(* IEC 61131-3 sources: xpxp/deepseek-coder-6.7b, 22 files *)

(* ---- 18.st ---- *)
plc
FUNCTION FC1003
	VAR_INPUT
		IN_R : REAL; (* Input real number *)
		IN_MAX, IN_MIN : REAL; (* Input min/max range for conversion *)
		OUT_MAX, OUT_MIN : REAL; (* Output min/max range for conversion *)
	END_VAR

	VAR_OUTPUT
		OUT_R : REAL; (* Result real number *)
		FEH : BOOL; (* Error flag indicating out-of-range *)
	END<｜begin▁of▁sentence｜>END_VAR

	VAR_TEMP
		DIFF1, DIFF2 : REAL; (* Temporary variables for scale calculation *)
		scl_factor : REAL; (* Scaling factor *)
		rescaled : REAL; (* Input rescaled to original range *)
	END<｜begin▁of▁sentence｜>END_VAR

	// Calculate scaling factor
	scl_factor := (OUT_MAX - OUT_MIN) / (IN_MAX - IN_MIN);

	// Rescale input value from its original range into the new one
	rescaled := scl_factor * (IN_R - IN_MIN) + OUT_MIN;

	(* Check if result is within output range *)
	IF ((rescaled < OUT_MIN) OR (rescaled > OUT_MAX)) THEN
		// If not, set error flag and return
		FEH := TRUE;
	ELSE
		OUT_R := rescaled;
	END_IF;

	// Return result and error flag to caller
	RETURN;
END_FUNCTION

(* ---- 22.st ---- *)
PLC_Programming
FUNCTION BLOCK fbMoveArm
VAR_INPUT
	MoveToWorkCmd : BOOL; // Move towards Work position command
	MoveToHomeCmd : BOOL; // Move towards Home position command
	AtWorkSensor : BOOL;  // Sensor indicating the arm is at the Work position
	AtHomeSensor : BOOL;  // Sensor indicating the arm is at the Home position
	MovementPermitted : BOOL; // Global safety signal allowing movement
END_VAR

VAR_OUTPUT
	MotorForward : BOOL; // Controls motor to move towards Work position
	MotorReverse : BOOL; // Controls motor to move towards Home position
END_VAR

// Store the previous command status for cancellation logic
VAR
	PrevMoveToWorkCmd : BOOL;
	PrevMoveToHomeCmd : BOOL;
END_VAR

IF MovementPermitted THEN
	// Cancel movement in opposite direction if current command is pressed
	MotorForward := (NOT PrevMoveToHomeCmd) AND MoveToWorkCmd;
	MotorReverse := (NOT PrevMoveToWorkCmd) AND MoveToHomeCmd;

	// Remember the status of current commands for cancellation logic
	PrevMoveToWorkCmd := MoveToWorkCmd;
	PrevMoveToHomeCmd := MoveToHomeCmd;
ELSE // If movement is not permitted, stop motors immediately
	MotorForward := FALSE;
	MotorReverse := FALSE;
END_IF

// Stop motor if at the target position
MotorForward := MotorForward AND (NOT AtWorkSensor);
MotorReverse := MotorReverse AND (NOT AtHomeSensor);
END_FUNCTION_BLOCK

(* ---- 1.st ---- *)
plc
PROGRAM MyProgram
VAR
    // Global Variables
	xAllOn : BOOL;
	xAlarm1: BOOL := FALSE;
	xAlarm2: BOOL := FALSE;
	xAllOff: BOOL;
END_VAR

// Initialize your variables here (if any)
// For example, xAllOn := TRUE;

FUNCTION_BLOCK FbUpdateAlarms
VAR_INPUT
    inAlarm1: BOOL;
    inAlarm2: BOOL;
END_VAR
VAR_OUTPUT
    outAlarm1 : BOOL;
    outAlarm2 : BOOL;
END_VAR
BEGIN
    // Update the alarms based on the input values
    IF (inAlarm1 = TRUE) THEN
        outAlarm1 := TRUE;
    END_IF;

    IF (inAlarm2 = TRUE) THEN
        outAlarm2 := TRUE;
    END_IF;
END_FUNCTION_BLOCK

// Create a new FB for updating alarms
FbUpdateAlarms(xAllOn, xAllOff, xAlarm1, xAlarm2);

(* ---- 11.st ---- *)
plc
PROGRAM SignFunction
VAR
    x : REAL; // input variable
END_VAR

FUNCTION_BLOCK FB_Sign
VAR_INPUT
    a : REAL;
END_VAR

VAR_OUTPUT
    result : INT;
END_VAR
END_FUNCTION_BLOCK

// Main function block where the program starts
FUNCTION_BLOCK FB_Main
VAR_INPUT
    x : REAL; // input variable
END_VAR

VAR_OUTPUT
    signValue : INT;
END_VAR
END_FUNCTION_BLOCK

(* ---- 19.st ---- *)
plaintext
PROGRAM Program1

FUNCTION_BLOCK FB1005
    (* VARIABLES DECLARATION *)
    VAR_INPUT
        START : BOOL;   // Start input for measurement cycle
        DICKE, V_MAX, V_MIN: REAL;  // Plate thickness and tolerance band values
    END_VAR

    VAR_OUTPUT
        D_MAX, D_MIN: REAL;  // Outputs for the maximum (D_MAX) and minimum (D_MIN) plate thickness
        P1: BOOL;   // Reject light P1 output
    END_VAR

    VAR
        FO: BOOL;  // Flag to indicate if a measurement is currently ongoing
        M_MAX, M_MIN : REAL;  // Maximum and minimum plate thickness during measurement cycle
    END_VAR
END_FUNCTION_BLOCK

(* FUNCTION BLOCK IMPLEMENTATION *)
PROGRAM Main
BEGIN
    (* Initialization of function block FB1005 *)
    FB1005(START := FALSE, DICKE := 0.0, V_MAX := 0.0, V_MIN := 0.0);

    (* Program main loop *)
    WHILE TRUE DO
        IF FB1005.START = TRUE THEN
            FO := TRUE;   // Start a measurement cycle

            M_MAX := DICKE;  // Initialize maximum plate thickness to current measured value
            M_MIN := DICKE;  // Initialize minimum plate thickness to current measured value
        END_IF;

        IF FO = TRUE THEN    // If a measurement cycle is ongoing
            FB1005.D_MAX := M_MAX;   // Output the maximum plate thickness
            FB1005.D_MIN := M_MIN;   // Output the minimum plate thickness

            IF (M_MAX > V_MAX) OR (M_MIN < V_MIN) THEN  // If current measurement violates tolerance band
                FB1005.P1 := TRUE;    // Switch on reject light P1
            END_IF;
        ELSE   // Else if no measurement cycle is ongoing, reset outputs
            FB1005.D_MAX := 0.0;
            FB1005.D_MIN := 0.0;
            FB1005.P1 := FALSE;
        END_IF;

        // Update maximum and minimum plate thickness for next measurement cycle
        M_MAX := MAX(M_MAX, DICKE);
        M_MIN := MIN(M_MIN, DICKE);
    END_WHILE;
END PROGRAM

(* ---- 20.st ---- *)
plaintext
PROGRAM MyProgram
VAR
    // Instantiate our interlock function block
    InterlockFb : INTERLOCK;

    // Declare the inputs I1, I2 and TL
    I1 : BOOL;
    I2 : BOOL;
    TL : TIME := T#5s;  // Dead time of 5 seconds
END_VAR

FUNCTION_BLOCK INTERLOCK
    VAR_INPUT
        I1 : BOOL;
        I2 : BOOL;
        TL : TIME;
    END_VAR

    VAR_OUTPUT
        Q1 : BOOL;
        Q2 : BOOL;
    END_VAR

    VAR
        T1 : TOF; // Time of FAlse for Q1
        T2 : TOF; // Time of False for Q2
    END_VAR

    IF I1 AND NOT Q1 THEN // If input is TRUE and output is FALSE, set Q1 to TRUE after dead time TL
        Q1(PT:=TL);
    ELSE
        Q1 := FALSE; // Reset Q1 if inputs are FALSE or already at TRUE for longer than deadtime TL
    END_IF;

    IF I2 AND NOT Q2 THEN // Same logic applies to Q2
        Q2(PT:=TL);
    ELSE
        Q2 := FALSE;
    END_IF;
END_FUNCTION_BLOCK

// Connections between PLC inputs and FB variables
I1 := DI[0]; // Connecting a digital input DI[0] to I1
I2 := DI[1]; // Connecting another digital input DI[1] to I2

InterlockFb(I1:=I1, I2:=I2, TL:=TL);  // Instantiating the FB in a way that its inputs correspond to our declared variables

Q1 := InterlockFb.Q1;  // Connecting the output Q1 of the function block back to an output on the PLC
Q2 := InterlockFb.Q2;  // Same logic applies for Q2
END_PROGRAM

(* ---- 21.st ---- *)
plc
FUNCTION_BLOCK BURNER
VAR_INPUT
    IN  : BOOL;
    STAGE2  : BOOL;
    OVER_TEMP  : BOOL;
    OIL_TEMP : BOOL := TRUE;
    FLAME  : BOOL;
    RST  : BOOL;
    RST_TIMER  : BOOL;
    PRE_HEAT_TIME  : TIME := t#5s;
    PRE_VENT_TIME : TIME := t#15s;
    PRE_IGNITE_TIME  : TIME := t#15s;
    POST_IGNITE_TIME  : TIME := t#25s;
    STAGE2_DELAY : TIME := t#10s;
    SAFETY_TIME  : TIME := t#5s;
    LOCKOUT_TIME : TIME := t#10s;
    MULTIPLE_IGNITION  : BOOL := TRUE;
    KW1  : REAL;
    KW2  : REAL;
END_VAR
VAR_OUTPUT
    MOTOR  : BOOL;
    COIL1  : BOOL;
    COIL2  : BOOL;
    PRE_HEAT  : BOOL;
    IGNITE  : BOOL;
    FAIL  : BOOL;
    KWH : REAL;
    STATUS  : BYTE;
END_VAR
VAR_IN_OUT
    RUNTIME1  : UDINT;
    RUNTIME2  : UDINT;
    CYCLES  : UDINT;
END_VAR
VAR
    state  : INT := 0; (* State variable to hold the current state of BURNER *)
    last  : TIME; (* Last cycle time *)
    tx  : TIME; (* Timeout *)
    last_change  : TIME; (* Last change in input *)
    timer1  : TON; (* Timer for PRE_HEAT_TIME *)
    timer2  : TON; (* Timer for other times *)
    oil_temp_last  : BOOL; (* Last state of OIL_TEMP *)
    cycles2  : UDINT; (* Number of cycles since RST was TRUE *)
END_VAR
END_FUNCTION_BLOCK

(* ---- 10.st ---- *)
plc
PROGRAM Sigmoid
VAR
    // Input variable for input data X
    input : REAL; END_VAR

    // Output variable for result Y
    output : REAL; END_VAR
END_VAR
    // Variables used in the sigmoid calculation
    temp1, temp2: REAL;
    numerator: LREAL;
    denominator: LREAL;

BEGIN
    // Calculation of sigmoid value
    temp1 := EXP(input);
    temp2 := 1 + temp1;

    numerator := temp1;
    denominator := temp2 * temp2;

    output := numerator / denominator;
END_PROGRAM

(* ---- 12.st ---- *)
plc
PROGRAM HyperbolicSine
    VAR
        X : REAL; (* Input variable *)
        Temp1, Temp2 : REAL; (* Temporary variables to hold intermediate results *)
        Result : REAL; (* Output variable for the result *)
    END_VAR

    (* Hyperbolic Sine Function using Exponential Function *)
    HSINE := EXP(X) / (EXP(X) + EXP(-X)) * 2.0;
END_PROGRAM

(* ---- 13.st ---- *)
plc
PROGRAM MainProgram
VAR
    aNumbers: ARRAY [0..99] OF INT := [123, 456, 789, ...]; (* Array of random numbers *)
    nCnt: INT;                                         (* Loop counter *)
END_VAR

BEGIN
    FOR nCnt := 0 TO MAXNUMBERS DO                      (* Initialize array with random values *)
        aNumbers[nCnt] := RANDOM(1, 5000);
    END_FOR

    nCnt := 0;                                          (* Reset counter for loop *)

    REPEAT                                            (* Loop to search for number *)
        IF aNumbers[nCnt] = 10 THEN                     (* Abort condition 1: found the number *)
            EXIT;
        END_IF

        IF nCnt = MAXNUMBERS THEN                       (* Abort condition 2: reached end of list *)
            EXIT;
        END_IF

        nCnt := nCnt + 1;                              (* Increment counter *)
    UNTIL
        TRUE;                                           (* This is always true, so the loop will exit when one of the conditions are met *)
    END_REPEAT

    IF aNumbers[nCnt] <> 10 AND nCnt <> MAXNUMBERS THEN(* Check if we exited due to reaching end of list *)
        (* Number 10 not found in array, do something else. e.g., Display message *)
        PRINT 'Number 10 was not found.'
    END_IF;
END_PROGRAM

(* ---- 14.st ---- *)
plc
PROGRAM Program0
VAR_GLOBAL
    MEW : REAL; // Measured External Working Value (input)
    SP : REAL;  // Set Point (predetermined value to switch on/off OUT)
    HYS : REAL; // Hysteresis in % of SP (predetermined value)
    OUT : BOOL; // Output (output)
END_VAR

FUNCTION FC1001 : BOOL
// This function compares MEW with SP considering the hysteresis.
// If MEW is within HYS% of SP, the function returns TRUE else FALSE.
VAR
    P_HYS: REAL; // Proportional Hysteresis Value
END_VAR
BEGIN
    // Calculate the proportional hysteresis value
    P_HYS := SP * (1 + HYS/100);

    // Compare MEW with the set point considering the hysteresis
    IF (MEW >= (SP - P_HYS)) AND (MEW <= (SP + P_HYS)) THEN
        FC1001 := TRUE; // Return TRUE if MEW is within SP ± HYS%
    ELSE
        FC1001 := FALSE; // Else return FALSE
    END_IF;
END_FUNCTION

PROGRAM main (*TODO: Add your comment *)
BEGIN
   // Initialisation of variables.
   MEW := 0.0;
   SP := 50.0;
   HYS := 10.0;

   OUT := FC1001(MEW,SP,HYS); // Invoke the function and assign its return value to OUT variable.
END_PROGRAM

(* ---- 15.st ---- *)
plc
PROGRAM FC1002
VAR_INPUT
	E_A, SENSOR: BOOL; // Input switch and sensor states
END_VAR
VAR
	ZEIT:TON; // Timer to measure time
	ALARM :BOOL; // Flag for alarm state
	TEMP_HU, TEMP_AL:BOOL; // Temporary variables for P_HU and P_AL
END_VAR
VAR_OUTPUT
	P_HU, P_AL: BOOL; // Output states of horn and alarm
END_VAR
BEGIN
	// Initialize the timer and output states at start
	ZEIT(IN:= E_A);
	TEMP_HU := FALSE;
	TEMP_AL := FALSE;

	// Check if sensor detects approaching object or person
	IF SENSOR = TRUE THEN
		// If detected, turn on TEMP_HU and start timer
		TEMP_HU := TRUE;
		ZEIT(P:= TRUE);

		// Turn off alarm if exists
		TEMP_AL := FALSE;

		// Check if the detection persists for more than 3 seconds
		IF ZEIT.Q THEN
			TEMP_HU := FALSE; // If yes, turn off TEMP_HU
			TEMP_AL := TRUE; // and activate alarm
		END_IF
	ELSE // If no detection, reset timer and alarm (if any)
		ZEIT(P:= FALSE);
		TEMP_AL := FALSE;
	END_IF;

	// Assign temporary variables to output states
	P_HU := TEMP_HU;
	P_AL := TEMP_AL;
END_PROGRAM

(* ---- 16.st ---- *)
plaintext
PROGRAM TrafficLightProgram
VAR
    // Inputs
	VAR_INPUT
        Timer : UDINT; (* Global timer, should be running and updating every 1ms *)
    END_VAR

    VAR_OUTPUT
        North_green : BOOL;
        North_yellow : BOOL;
        North_red : BOOL;
        East_green : BOOL;
        East_yellow : BOOL;
        East_red : BOOL;
    END_VAR

END_VAR

IF Timer > 0 AND Timer < 500 THEN (* 1st cycle: North light is green, East light is red *)
    North_green := TRUE;
    North_yellow := FALSE;
    North_red := FALSE;
    East_green := FALSE;
    East_yellow := FALSE;
    East_red := TRUE;
ELSIF Timer > 500 AND Timer < 950 THEN (* 2nd cycle: Yellow light for North *)
    North_green := FALSE;
    North_yellow := TRUE;
    North_red := FALSE;
    East_green := FALSE;
    East_yellow := FALSE;
    East_red := TRUE;
ELSIF Timer > 950 AND Timer < 1000 THEN (* 3rd cycle: North light is red, East light is green *)
    North_green := FALSE;
    North_yellow := FALSE;
    North_red := TRUE;
    East_green := TRUE;
    East_yellow := FALSE;
    East_red := FALSE;
ELSIF Timer > 1000 AND Timer < 1500 THEN (* 4th cycle: Yellow light for East *)
    North_green := FALSE;
    North_yellow := FALSE;
    North_red := TRUE;
    East_green := FALSE;
    East_yellow := TRUE;
    East_red := FALSE;
ELSE (* Reset all lights at the end of cycle *)
    North_green := FALSE;
    North_yellow := FALSE;
    North_red := FALSE;
    East_green := FALSE;
    East_yellow := FALSE;
    East_red := TRUE;
END_IF;
END_PROGRAM

(* ---- 17.st ---- *)
PLC
PROGRAM WeatherStationProgram
VAR
    // Variables for temperature and humidity
    aiOutside : INT;   // Analog input for outside temperature
    aiHumidity: INT;  // Analog input for humidity

    // String variable to display the text message
    sShowText : STRING(80);
END_VAR

// Main program function
FUNCTION WeatherStationProgram : BOOL
BEGIN
    CASE aiOutside OF
        1..17:   sShowText := 'Cold';  // If temperature is below 18°C
        18..25:  sShowText := 'Opt';   // If temperature is between 18°C and 25°C
        ELSE:    sShowText := 'Hot';   // If temperature is above 25°C
    END_CASE

    CASE aiHumidity OF                   // Nested case for humidity
        40..75 WHEN EQUAL aiOutside:18..25, (OTHERS) : sShowText := 'Opt';  // If temperature is between 18°C and 25°C and humidity is between 40% and 75%, display "Opt"
        ELSE:                                  // Otherwise, for other cases of humidity and temperature
            CASE aiOutside OF
                1..17:   sShowText := 'Temp. OK';  // If temperature is below 18°C
                ELSE:    sShowText := 'Temp. OK';  // If temperature is above 25°C
            END_CASE
        (OTHERS) : sShowText := 'Invalid humidity input';   // For invalid humidity inputs
    END_CASE

    WeatherStationProgram := TRUE;
END_FUNCTION

(* ---- 2.st ---- *)
plc
PROGRAM BinomialCoefficient
    VAR_INPUT
        N : INT; // Total number of items
        K : INT; // Number of items to choose
        i : INT; // Loop counter
    END_VAR

    VAR
        result : LONG := 1; // Result will be stored here
    END_VAR

BEGIN
    FOR i := 1 TO (K) DO // From 1 to K, both inclusive
        result := result * ((N + i - K) DIV i); // Calculate n*(n-1)*...(n-k+1)/k
    END_FOR;
END_PROGRAM

(* ---- 3.st ---- *)
plc
PROGRAM FibonacciProgram
// Input variables
VAR_INPUT
    X : INT; // the number to calculate fibonacci for
END_VAR

// Internal variables
VAR
    t1 : DINT;
    t2 : DINT;
    x_tmp : INT;
END_VAR

BEGIN
    IF X > 0 THEN BEGIN
        // Base case for Fibonacci (F(0) = 0, F(1) = 1)
        t1 := 0;
        t2 := 1;

        FOR i:=2 TO X DO BEGIN   // Iterative calculation of fibonacci number
            x_tmp := t1 + t2;
            t1 := t2;
            t2 := x_tmp;
        END_FOR
    END
END_IF
END_PROGRAM

(* ---- 4.st ---- *)
plc
PROGRAM Program0
VAR
    VAR_INPUT  at %IX0.0 : INT; (* Analog input for fill level *)
    VAR_OUTPUT at %QX0.0 : BOOL; (* Output for low fill level *)
    VAR_OUTPUT at %QX0.1 : BOOL; (* Output for ok fill level *)
    VAR_OUTPUT at %QX0.2 : BOOL; (* Output for high fill level *)

    aiLevel  : INT;       (* Analog input value *)
    PercentLevel  : UINT; (* Fill level in percent *)
    doLow  : BOOL;        (* Low fill level output indicator *)
    doOk  : BOOL;         (* Ok fill level output indicator *)
    doHigh  : BOOL;       (* High fill level output indicator *)
    doAlarm  : BOOL;      (* Alarm sounder simulation *)
END_VAR

BEGIN_PROGRAM
    aiLevel := INT_TO_UINT(aiLevel);   (* Conversion from INT to UINT type *)

    PercentLevel := (aiLevel / 32767) * 100;   (* Convert the analog value to percent representation *)

    doAlarm := FALSE;   (* Initialize alarm indicator *)

    CASE PercentLevel OF
        0 .. 99: (* If fill level is below 1% *)
            doLow := TRUE;
            doOk := FALSE;
            doHigh := FALSE;
            doAlarm := TRUE;
        100 .. 254: (* If fill level is between 1% and 99.99% *)
            doLow := FALSE;
            doOk := TRUE;
            doHigh := FALSE;
            doAlarm := FALSE;
        255 .. 32767: (* If fill level is above 99.99% *)
            doLow := FALSE;<｜begin▁of▁sentence｜>
            doOk := FALSE;
            doHigh := TRUE;
            doAlarm := FALSE;
    END_CASE;
END_PROGRAM Program0

(* ---- 5.st ---- *)
plaintext
PROGRAM MyProgram
VAR
    VAR_INPUT
        Start_Loop : BOOL; // start the timer when this is false
        Sensed_Car : BOOL;
        Sensed_App : BOOL;
        Auth : STRING(10); // max length of 10 chars, adjust as necessary
    END_VAR

    VAR_OUTPUT
        Gate_Open : BOOL; // indicates whether the gate is open
        Close_Gate_Inst : BOOL; // set this to TRUE when you want to close the gate manually
    END_VAR

    CONSTANT
        my_defined_str : STRING(4) := 'abcd';
    END_CONSTANT

    VAR
        one_hour : TIME := T#1h; // time span of 1 hour
        One_Hour_Timer : TON; // timer that will reset after 1 hour
    END_VAR
END_PROGRAM

(* ---- 6.st ---- *)
plc
PROGRAM MyProgram
VAR
    (*-- digital outputs*)
    doConvTop: BOOL;
    doConvBottom: BOOL;
    doConvLift: BOOL;
    doLiftTop: BOOL;
    doLiftBottom: BOOL;
    doLiftUnload: BOOL;

    (*-- digital inputs*)
    diConvTop: BOOL;
    diConvBottom: BOOL;
    diLiftTop: BOOL;
    diLiftBottom: BOOL;
    diLiftUnload: BOOL;
    diBoxLift: BOOL;

    (*-- status variables*)
    selectLift: UINT := WAIT;
    ConvTopOn: BOOL := FALSE;
    ConvBottomOn: BOOL := FALSE;
END_VAR

BEGIN
    CASE selectLift OF
        WAIT:
            (* Wait for lift request *)
            IF diConvTop OR diConvBottom THEN // if any of the conveyors are activated, stop them and move to requested position
                ConvTopOn := FALSE;
                doConvTop := FALSE;

                ConvBottomOn := FALSE;
                doConvBottom := FALSE;

                IF diConvTop THEN // if top conveyor is activated, go to bottom and vice versa
                    selectLift := BOTTOM_POSITION;
                ELSE
                    selectLift := TOP_POSITION;
                END_IF
            END_IF
        TOP_POSITION:
            (* Lift at top position *)
            IF NOT diConvTop THEN // if the conveyor is deactivated, stop it and start moving to unload position
                doLiftUnload := TRUE;

                ConvBottomOn := FALSE;
                doConvBottom := FALSE;

                selectLift := UNLOAD_POSITION; // change state to unloading position
            END_IF
        BOTTOM_POSITION:
            (* Lift at bottom position *)
            IF NOT diConvBottom THEN // if the conveyor is deactivated, stop it and start moving to unload position
                doLiftUnload := TRUE;

                ConvTopOn := FALSE;
                doConvTop := FALSE;

                selectLift := UNLOAD_POSITION; // change state to unloading position
            END_IF
        UNLOAD_POSITION:
            (* Lift at unload position *)
            IF diBoxLift THEN // if box is in lift, start moving back to initial positions
                doConvLift := FALSE;

                selectLift := WAIT; // change state to waiting for requests
            END_IF
    END_CASE;
END_PROGRAM

(* ---- 7.st ---- *)
plc
PROGRAM MyProgram
VAR
    // Array declaration
    aWeights : ARRAY[0..4] OF INT;

    // Counter variable
    iCnt : USINT;

    // Summation and average variables
    sumWeight : LINT;
    avgWeight : INT;
END_VAR

FUNCTION CalculateAverage: INT
    VAR
        tempSum : LINT;
    END_VAR

    tempSum := 0;
    FOR iCnt := 0 TO 4 DO // Iterating over the array elements
        tempSum += aWeights[iCnt]; // Adding up all weights
    END_FOR

    CalculateAverage := tempSum / 5; // Calculating average weight
END_FUNCTION

// Main program function
FUNCTION _Main : BOOL
BEGIN
    // Assuming aWeights array is filled with some values at the beginning of this function
   avgWeight := CalculateAverage(); // Calling our function and storing result in avgWeight variable
END_FUNCTION

(* ---- 8.st ---- *)
plaintext
PROGRAM Program01
VAR_INPUT
    X : REAL; // Input variable
END_VAR

VAR
    w : REAL; // Lambert W function value (output)
    i : INT;  // Loop counter for Newton-Raphson method
    we, w1e, ewx : REAL; // Intermediate variables in the Newton-Raphson method
    last : DWORD; // Used to ensure convergence of Newton-Raphson method (prevent infinite loop)
END_VAR

FUNCTION LambertW : REAL
    VAR_INPUT
        x : REAL;
    END_VAR

    LambertW := XYZ; (* Placeholder function, this should return the value of Lambert W function for input 'x' *)
END_FUNCTION

PROGRAM MainProgram
BEGIN
    FOR i := 1 TO 100 DO // Iterate up to a maximum of 100 steps in Newton-Raphson method, or until convergence is reached
        we := LambertW(X);
        ewx := EXP(we) * X;

        IF (ABS(ewx - 1.0) < 0.00001) THEN // Check for convergence based on difference between actual value and expected value of w*e^w
            w := we;
            EXIT;
        END_IF

        w1e := 1.0 + we / ewx;

        IF (ABS(w - w1e) < 0.00001) THEN // Check for convergence based on difference between two consecutive values of Lambert W function approximation
            w := w1e;
            EXIT;
        END_IF

        w := w1e; // Update the value of w
    END_FOR
END_PROGRAM

(* ---- 9.st ---- *)
plc
PROGRAM LeapYearProgram
VAR
    YEAR : INT; (* Input Variable *)
    IS_LEAP : BOOL; (* Output Variable to indicate whether the input year is a leap year or not *)
END_VAR

FUNCTION CheckLeapYear: BOOL (* Function to check if a given year is a leap year *)
VAR_INPUT
    YearToCheck : INT; (* The year to check *)
END_VAR
VAR
    DivisibleBy4 : BOOL; (* Indicates whether the year can be divided by 4 without a remainder *)
    DivisibleBy100 : BOOL; (* Indicates whether the year can be divided by 100 without a remainder *)
    DivisibleBy400 : BOOL; (* Indicates whether the year can be divided by 400 without a remainder *)
END_VAR
BEGIN
    DivisibleBy4 := YearToCheck MOD 4 = 0; (* Check if divisible by 4 *)
    DivisibleBy100 := YearToCheck MOD 100 = 0; (* Check if divisible by 100 *)
    DivisibleBy400 := YearToCheck MOD 400 = 0; (* Check if divisible by 400 *)

    IF DivisibleBy4 THEN (* If the year can be divided by 4, then it's a leap year unless: *)
        IF NOT DivisibleBy100 OR DivisibleBy400 THEN (* - It can also be divided by 100 but not by 400 *)
            CheckLeapYear := TRUE; (* Then it is a leap year. *)
        ELSE (* Otherwise, it's not a leap year *)
            CheckLeapYear := FALSE;
        END_IF;
    ELSE (* If the year cannot be divided by 4, then it's not a leap year *)
        CheckLeapYear := FALSE;
    END_IF;
END_FUNCTION

(* Main program part to use the function and set the output variable according to its return value *)
BEGIN
    IS_LEAP := CheckLeapYear(YEAR); (* Calling the function with input year and storing its result in IS_LEAP *)
END_PROGRAM
